// TIA Portal V20 export
// export: Created 2026-04-20T18:50:18.2063652Z, ExportSetting WithDefaults, DisplayName Totally Integrated Automation Portal, DisplayVersion V20, DisplayName TIA Portal Openness, DisplayVersion V20, DisplayName TIA Portal Version Control Interface, DisplayVersion V20, DisplayName STEP 7 Professional, DisplayVersion V20, DisplayName STEP 7 Safety, DisplayVersion V20, DisplayName WinCC Basic/Comfort/Advanced, DisplayVersion V20
TYPE "UDT_ControlValve"
// stored: IsFailsafeCompliant false
   STRUCT
      valveTag : String[16] := 'V-000';   // P and ID tag reference (e.g. V-10101)
      valveType : Int := 1;   // Mechanical type: 1=Ball 2=Butterfly 3=Diaphragm 4=Globe 5=Needle
      travelTime { S7_SetPoint := 'True'} : Time := T#4S;   // Full stroke travel time
      positionSetpoint { S7_SetPoint := 'True'} : Real := 0.0;   // Commanded position in percent (0 = closed, 100 = open)
      deadband { S7_SetPoint := 'True'} : Real := 1.5;   // Position deadband in percent to reduce actuator wear
      flowLimits { S7_SetPoint := 'True'} : "UDT_AlarmLimits";   // Alarm limits for the flow measurement
      pressureLimits { S7_SetPoint := 'True'} : "UDT_AlarmLimits";   // Alarm limits for the pressure measurement
      comment : String[64] := '';   // Free text notes for commissioning
   END_STRUCT;
END_TYPE
